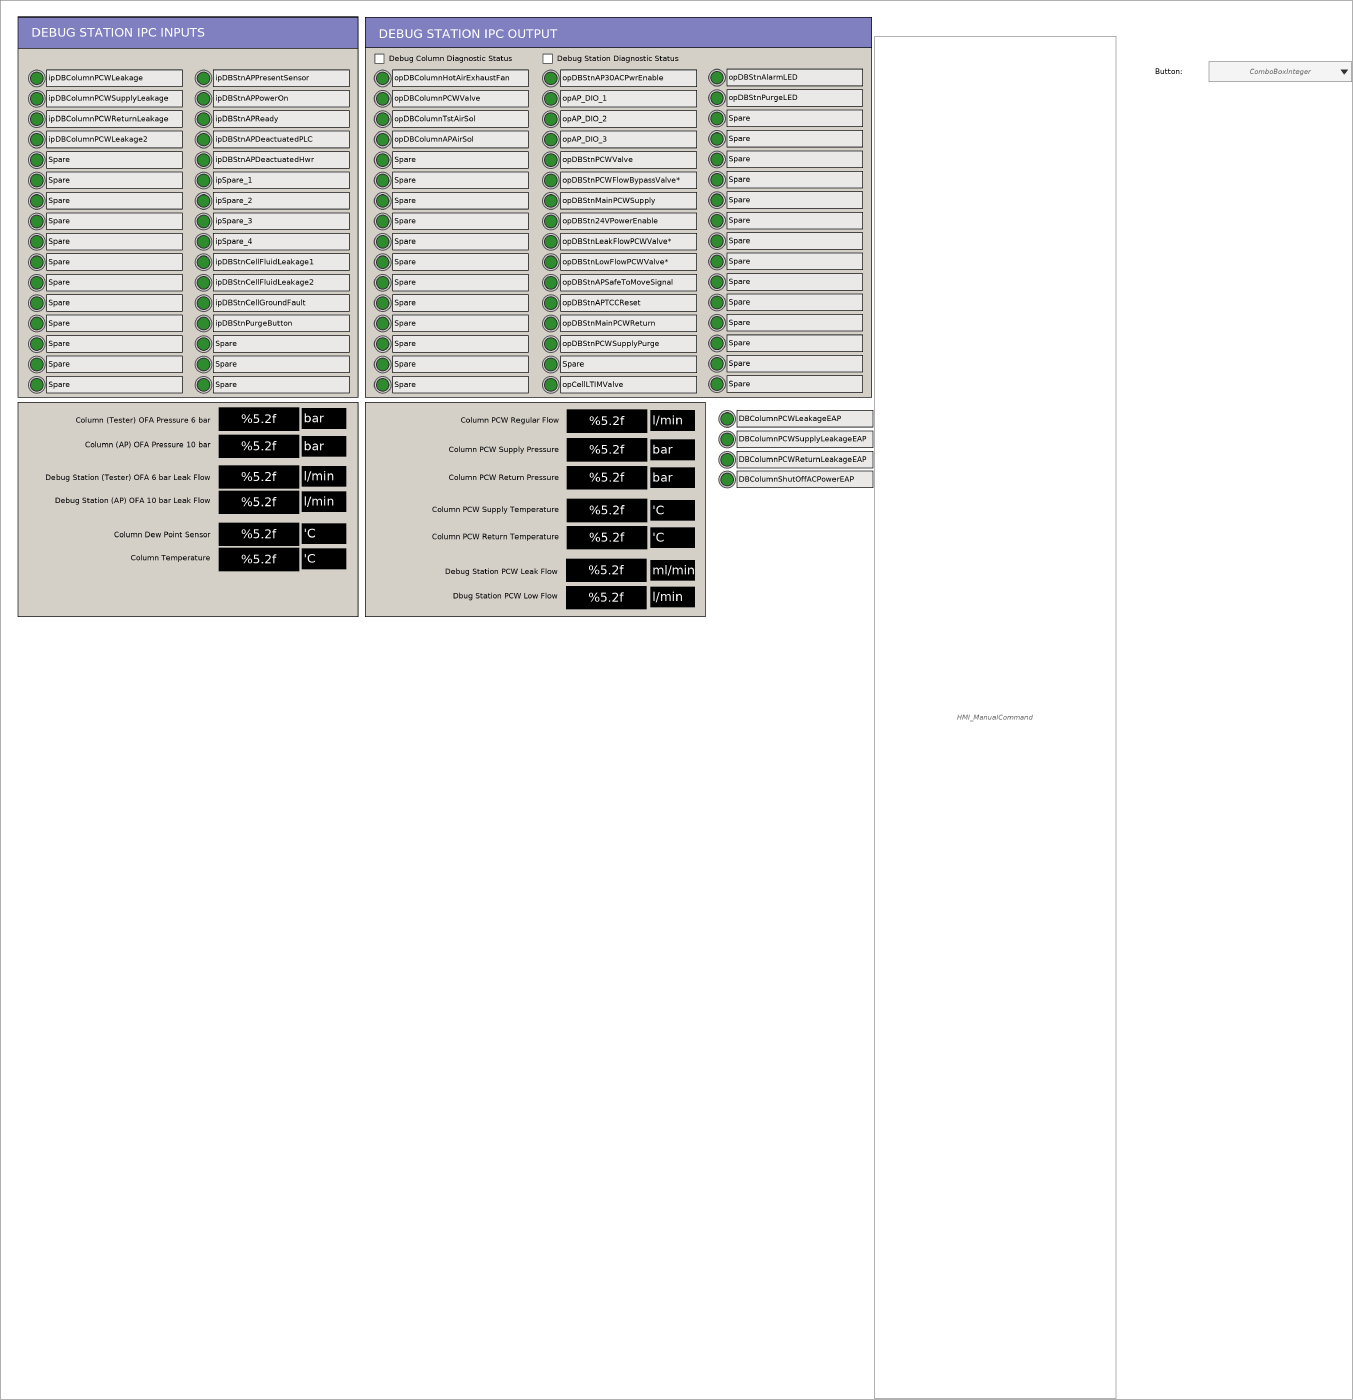
VISUALIZATION HMI_DebugStation  // 1987x2055
    Rectangle (536,590 500x315)
    Rectangle (26,590 500x315)
    Rectangle (536,42 744x541)
    Rectangle (536,25 744x45)
    Label (553,30 500x40), "DEBUG STATION IPC OUTPUT"
    Rectangle (26,24 500x559)
    Rectangle (26,25 500x46)
    Label (43,28 500x40), "DEBUG STATION IPC INPUTS"
    RoundedRectangle (68,102 200x25), "ipDBColumnPCWLeakage"
    Lamp1 (39,100 30x30), variable: fbDebugColumn.stDebugColumnDIO.ipDBColumnPCWLeakage, style: Lamp-Lamp1-Green
    RoundedRectangle (576,102 200x25), "opDBColumnHotAirExhaustFan"
        toggle fbDebugColumn.stDebugColumnDIO.opDBColumnHotAirExhaustFan
    Lamp1 (547,100 30x30), variable: fbDebugColumn.stDebugColumnDIO.opDBColumnHotAirExhaustFan, style: Lamp-Lamp1-Green
    RoundedRectangle (68,132 200x25), "ipDBColumnPCWSupplyLeakage"
    Lamp1 (39,130 30x30), variable: fbDebugColumn.stDebugColumnDIO.ipDBColumnPCWSupplyLeakage, style: Lamp-Lamp1-Green
    RoundedRectangle (68,162 200x25), "ipDBColumnPCWReturnLeakage"
    Lamp1 (39,160 30x30), variable: fbDebugColumn.stDebugColumnDIO.ipDBColumnPCWReturnLeakage, style: Lamp-Lamp1-Green
    RoundedRectangle (68,192 200x25), "ipDBColumnPCWLeakage2"
    Lamp1 (39,190 30x30), variable: fbDebugColumn.stDebugColumnDIO.ipDBColumnPCWLeakage2, style: Lamp-Lamp1-Green
    RoundedRectangle (68,222 200x25), "Spare"
    Lamp1 (39,220 30x30), style: Lamp-Lamp1-Green
    RoundedRectangle (68,252 200x25), "Spare"
    Lamp1 (39,250 30x30), style: Lamp-Lamp1-Green
    RoundedRectangle (68,282 200x25), "Spare"
    Lamp1 (39,280 30x30), style: Lamp-Lamp1-Green
    RoundedRectangle (68,312 200x25), "Spare"
    Lamp1 (39,310 30x30), style: Lamp-Lamp1-Green
    RoundedRectangle (68,342 200x25), "Spare"
    Lamp1 (39,340 30x30), style: Lamp-Lamp1-Green
    RoundedRectangle (68,372 200x25), "Spare"
    Lamp1 (39,370 30x30), style: Lamp-Lamp1-Green
    RoundedRectangle (68,402 200x25), "Spare"
    Lamp1 (39,400 30x30), style: Lamp-Lamp1-Green
    RoundedRectangle (68,432 200x25), "Spare"
    Lamp1 (39,430 30x30), style: Lamp-Lamp1-Green
    RoundedRectangle (68,462 200x25), "Spare"
    Lamp1 (39,460 30x30), style: Lamp-Lamp1-Green
    RoundedRectangle (68,492 200x25), "Spare"
    Lamp1 (39,490 30x30), style: Lamp-Lamp1-Green
    RoundedRectangle (68,522 200x25), "Spare"
    Lamp1 (39,520 30x30), style: Lamp-Lamp1-Green
    RoundedRectangle (68,552 200x25), "Spare"
    Lamp1 (39,550 30x30), style: Lamp-Lamp1-Green
    RoundedRectangle (576,132 200x25), "opDBColumnPCWValve"
        toggle fbDebugColumn.stDebugColumnDIO.opDBColumnPCWValve
    Lamp1 (547,130 30x30), variable: fbDebugColumn.stDebugColumnDIO.opDBColumnPCWValve, style: Lamp-Lamp1-Green
    RoundedRectangle (576,162 200x25), "opDBColumnTstAirSol"
        toggle fbDebugColumn.stDebugColumnDIO.opDBColumnTstAirSol
    Lamp1 (547,160 30x30), variable: fbDebugColumn.stDebugColumnDIO.opDBColumnTstAirSol, style: Lamp-Lamp1-Green
    RoundedRectangle (576,192 200x25), "opDBColumnAPAirSol"
        toggle fbDebugColumn.stDebugColumnDIO.opDBColumnAPAirSol
    Lamp1 (547,190 30x30), variable: fbDebugColumn.stDebugColumnDIO.opDBColumnAPAirSol, style: Lamp-Lamp1-Green
    RoundedRectangle (576,222 200x25), "Spare"
    Lamp1 (547,220 30x30), style: Lamp-Lamp1-Green
    RoundedRectangle (576,252 200x25), "Spare"
    Lamp1 (547,250 30x30), style: Lamp-Lamp1-Green
    RoundedRectangle (576,282 200x25), "Spare"
    Lamp1 (547,280 30x30), style: Lamp-Lamp1-Green
    RoundedRectangle (576,312 200x25), "Spare"
    Lamp1 (547,310 30x30), style: Lamp-Lamp1-Green
    RoundedRectangle (576,342 200x25), "Spare"
    Lamp1 (547,340 30x30), style: Lamp-Lamp1-Green
    RoundedRectangle (576,372 200x25), "Spare"
    Lamp1 (547,370 30x30), style: Lamp-Lamp1-Green
    RoundedRectangle (576,402 200x25), "Spare"
    Lamp1 (547,400 30x30), style: Lamp-Lamp1-Green
    RoundedRectangle (576,432 200x25), "Spare"
    Lamp1 (547,430 30x30), style: Lamp-Lamp1-Green
    RoundedRectangle (576,462 200x25), "Spare"
    Lamp1 (547,460 30x30), style: Lamp-Lamp1-Green
    RoundedRectangle (576,492 200x25), "Spare"
    Lamp1 (547,490 30x30), style: Lamp-Lamp1-Green
    RoundedRectangle (576,522 200x25), "Spare"
    Lamp1 (547,520 30x30), style: Lamp-Lamp1-Green
    RoundedRectangle (576,552 200x25), "Spare"
    Lamp1 (547,550 30x30), style: Lamp-Lamp1-Green
    RoundedRectangle (313,102 200x25), "ipDBStnAPPresentSensor"
    Lamp1 (284,100 30x30), variable: stDebugStation.fbDBStnSeq.stDebugStationDIO.ipDBStnAPPresentSensor, style: Lamp-Lamp1-Green
    RoundedRectangle (313,132 200x25), "ipDBStnAPPowerOn"
    Lamp1 (284,130 30x30), variable: stDebugStation.fbDBStnSeq.stDebugStationDIO.ipDBStnAPPowerOn, style: Lamp-Lamp1-Green
    RoundedRectangle (313,162 200x25), "ipDBStnAPReady"
    Lamp1 (284,160 30x30), variable: stDebugStation.fbDBStnSeq.stDebugStationDIO.ipDBStnAPReady, style: Lamp-Lamp1-Green
    RoundedRectangle (313,192 200x25), "ipDBStnAPDeactuatedPLC"
    Lamp1 (284,190 30x30), variable: stDebugStation.fbDBStnSeq.stDebugStationDIO.ipDBStnHandlerSafeToEnterPLC, style: Lamp-Lamp1-Green
    RoundedRectangle (313,222 200x25), "ipDBStnAPDeactuatedHwr"
    Lamp1 (284,220 30x30), variable: stDebugStation.fbDBStnSeq.stDebugStationDIO.ipDBStnHandlerSafeToEnterHwr, style: Lamp-Lamp1-Green
    RoundedRectangle (313,252 200x25), "ipSpare_1"
    Lamp1 (284,250 30x30), variable: stDebugStation.fbDBStnSeq.stDebugStationDIO.ipSpare_1, style: Lamp-Lamp1-Green
    RoundedRectangle (313,282 200x25), "ipSpare_2"
    Lamp1 (284,280 30x30), variable: stDebugStation.fbDBStnSeq.stDebugStationDIO.ipSpare_2, style: Lamp-Lamp1-Green
    RoundedRectangle (313,312 200x25), "ipSpare_3"
    Lamp1 (284,310 30x30), variable: stDebugStation.fbDBStnSeq.stDebugStationDIO.ipSpare_3, style: Lamp-Lamp1-Green
    RoundedRectangle (313,342 200x25), "ipSpare_4"
    Lamp1 (284,340 30x30), variable: stDebugStation.fbDBStnSeq.stDebugStationDIO.ipSpare_4, style: Lamp-Lamp1-Green
    RoundedRectangle (313,372 200x25), "ipDBStnCellFluidLeakage1"
    Lamp1 (284,370 30x30), variable: stDebugStation.fbDBStnSeq.stDebugStationDIO.ipDBStnCellFluidLeakage1, style: Lamp-Lamp1-Green
    RoundedRectangle (313,402 200x25), "ipDBStnCellFluidLeakage2"
    Lamp1 (284,400 30x30), variable: stDebugStation.fbDBStnSeq.stDebugStationDIO.ipDBStnCellFluidLeakage2, style: Lamp-Lamp1-Green
    RoundedRectangle (313,432 200x25), "ipDBStnCellGroundFault"
    Lamp1 (284,430 30x30), variable: stDebugStation.fbDBStnSeq.stDebugStationDIO.ipDBStnCellGroundFault, style: Lamp-Lamp1-Green
    RoundedRectangle (313,462 200x25), "ipDBStnPurgeButton"
    Lamp1 (284,460 30x30), variable: stDebugStation.fbDBStnSeq.stDebugStationDIO.ipDBStnPurgeButton, style: Lamp-Lamp1-Green
    RoundedRectangle (313,492 200x25), "Spare"
    Lamp1 (284,490 30x30), style: Lamp-Lamp1-Green
    RoundedRectangle (313,522 200x25), "Spare"
    Lamp1 (284,520 30x30), style: Lamp-Lamp1-Green
    RoundedRectangle (313,552 200x25), "Spare"
    Lamp1 (284,550 30x30), style: Lamp-Lamp1-Green
    RoundedRectangle (823,102 200x25), "opDBStnAP30ACPwrEnable"
        toggle stDebugStation.fbDBStnSeq.stDebugStationDIO.opDBStnAP240ACPwrEnable
    Lamp1 (794,100 30x30), variable: stDebugStation.fbDBStnSeq.stDebugStationDIO.opDBStnAP240ACPwrEnable, style: Lamp-Lamp1-Green
    RoundedRectangle (823,132 200x25), "opAP_DIO_1"
        toggle stDebugStation.fbDBStnSeq.stDebugStationDIO.opAP_DIO_1
    Lamp1 (794,130 30x30), variable: stDebugStation.fbDBStnSeq.stDebugStationDIO.opAP_DIO_1, style: Lamp-Lamp1-Green
    RoundedRectangle (823,162 200x25), "opAP_DIO_2"
        toggle stDebugStation.fbDBStnSeq.stDebugStationDIO.opAP_DIO_2
    Lamp1 (794,160 30x30), variable: stDebugStation.fbDBStnSeq.stDebugStationDIO.opAP_DIO_2, style: Lamp-Lamp1-Green
    RoundedRectangle (823,192 200x25), "opAP_DIO_3"
        toggle stDebugStation.fbDBStnSeq.stDebugStationDIO.opAP_DIO_3
    Lamp1 (794,190 30x30), variable: stDebugStation.fbDBStnSeq.stDebugStationDIO.opAP_DIO_3, style: Lamp-Lamp1-Green
    RoundedRectangle (823,222 200x25), "opDBStnPCWValve"
        toggle stDebugStation.fbDBStnSeq.stDebugStationDIO.opDBStnPCWValve
    Lamp1 (794,220 30x30), variable: stDebugStation.fbDBStnSeq.stDebugStationDIO.opDBStnPCWValve, style: Lamp-Lamp1-Green
    RoundedRectangle (823,252 200x25), "opDBStnPCWFlowBypassValve*"
        toggle stDebugStation.fbDBStnSeq.stDebugStationDIO.opDBStnPCWFlowBypassValve
    Lamp1 (794,250 30x30), variable: stDebugStation.fbDBStnSeq.stDebugStationDIO.opDBStnPCWFlowBypassValve, style: Lamp-Lamp1-Green
    RoundedRectangle (823,282 200x25), "opDBStnMainPCWSupply"
        toggle stDebugStation.fbDBStnSeq.stDebugStationDIO.opDBStnBypassAPAirSupplySol
    Lamp1 (794,280 30x30), variable: stDebugStation.fbDBStnSeq.stDebugStationDIO.opDBStnBypassAPAirSupplySol, style: Lamp-Lamp1-Green
    RoundedRectangle (823,312 200x25), "opDBStn24VPowerEnable"
        toggle stDebugStation.fbDBStnSeq.stDebugStationDIO.opDBStn24VPowerEnable
    Lamp1 (794,310 30x30), variable: stDebugStation.fbDBStnSeq.stDebugStationDIO.opDBStn24VPowerEnable, style: Lamp-Lamp1-Green
    RoundedRectangle (823,342 200x25), "opDBStnLeakFlowPCWValve*"
        toggle stDebugStation.fbDBStnSeq.stDebugStationDIO.opDBStnLeakFlowPCWValve
    Lamp1 (794,340 30x30), variable: stDebugStation.fbDBStnSeq.stDebugStationDIO.opDBStnLeakFlowPCWValve, style: Lamp-Lamp1-Green
    RoundedRectangle (823,372 200x25), "opDBStnLowFlowPCWValve*"
        toggle stDebugStation.fbDBStnSeq.stDebugStationDIO.opDBStnLowFlowPCWValve
    Lamp1 (794,370 30x30), variable: stDebugStation.fbDBStnSeq.stDebugStationDIO.opDBStnLowFlowPCWValve, style: Lamp-Lamp1-Green
    RoundedRectangle (823,402 200x25), "opDBStnAPSafeToMoveSignal"
        toggle stDebugStation.fbDBStnSeq.stDebugStationDIO.opDBStnAPSafeToEngage
    Lamp1 (794,400 30x30), variable: stDebugStation.fbDBStnSeq.stDebugStationDIO.opDBStnAPSafeToEngage, style: Lamp-Lamp1-Green
    RoundedRectangle (823,432 200x25), "opDBStnAPTCCReset"
        toggle stDebugStation.fbDBStnSeq.stDebugStationDIO.opDBStnAPTCCReset
    Lamp1 (794,430 30x30), variable: stDebugStation.fbDBStnSeq.stDebugStationDIO.opDBStnAPTCCReset, style: Lamp-Lamp1-Green
    RoundedRectangle (823,462 200x25), "opDBStnMainPCWReturn"
        toggle stDebugStation.fbDBStnSeq.stDebugStationDIO.opDBStnMainPCWReturn
    Lamp1 (794,460 30x30), variable: stDebugStation.fbDBStnSeq.stDebugStationDIO.opDBStnMainPCWReturn, style: Lamp-Lamp1-Green
    RoundedRectangle (823,492 200x25), "opDBStnPCWSupplyPurge"
        toggle stDebugStation.fbDBStnSeq.stDebugStationDIO.opDBStnPCWSupplyPurge
    Lamp1 (794,490 30x30), variable: stDebugStation.fbDBStnSeq.stDebugStationDIO.opDBStnPCWSupplyPurge, style: Lamp-Lamp1-Green
    RoundedRectangle (823,522 200x25), "Spare"
    Lamp1 (794,520 30x30), style: Lamp-Lamp1-Green
    RoundedRectangle (823,552 200x25), "opCellLTIMValve"
        toggle stDebugStation.fbDBStnSeq.stDebugStationDIO.opCellLTIMValve
    Lamp1 (794,550 30x30), variable: stDebugStation.fbDBStnSeq.stDebugStationDIO.opCellLTIMValve, style: Lamp-Lamp1-Green
    Textfield (320,597 120x36), "%5.2f", text variable: fbDebugColumn.stDebugColumnDIO.ipDBColumnTstAirPressure, input disabled if: TRUE
    Textfield (320,637 120x36), "%5.2f", text variable: fbDebugColumn.stDebugColumnDIO.ipDBColumnAPAirPressure, input disabled if: TRUE
    Textfield (320,682 120x36), "%5.2f", text variable: stDebugStation.fbDBStnSeq.stDebugStationDIO.ipDBStnTstAirLeakFlowSensor, input disabled if: TRUE
    Textfield (320,719 120x36), "%5.2f", text variable: stDebugStation.fbDBStnSeq.stDebugStationDIO.ipDBStnAPAirLeakFlowSensor, input disabled if: TRUE
    Label (51,686 261x30), "Debug Station (Tester) OFA 6 bar Leak Flow"
    Label (44,720 268x30), "Debug Station (AP) OFA 10 bar Leak Flow"
    Label (60,602 252x30), "Column (Tester) OFA Pressure 6 bar"
    Label (81,638 231x30), "Column (AP) OFA Pressure 10 bar"
    Textfield (830,819 120x36), "%5.2f", text variable: stDebugStation.fbDBStnSeq.stDebugStationDIO.ipDBStnPCWLeakFlowSensor, input disabled if: TRUE
    Textfield (830,859 120x36), "%5.2f", text variable: stDebugStation.fbDBStnSeq.stDebugStationDIO.ipDBStnPCWLowFlowSensor, input disabled if: TRUE
    Label (620,824 202x30), "Debug Station PCW Leak Flow"
    Label (574,860 248x30), "Dbug Station PCW Low Flow"
    Textfield (831,771 120x36), "%5.2f", text variable: fbDebugColumn.stDebugColumnDIO.ipDBColumnPCWReturnTemperature, input disabled if: TRUE
    Textfield (831,683 120x36), "%5.2f", text variable: fbDebugColumn.stDebugColumnDIO.ipDBColumnPCWReturnPressure, input disabled if: TRUE
    Textfield (831,600 120x36), "%5.2f", text variable: fbDebugColumn.stDebugColumnDIO.ipDBColumnPCWRegularFlowSensor, input disabled if: TRUE
    Textfield (831,642 120x36), "%5.2f", text variable: fbDebugColumn.stDebugColumnDIO.ipDBColumnPCWSupplyPressure, input disabled if: TRUE
    Textfield (831,731 120x36), "%5.2f", text variable: fbDebugColumn.stDebugColumnDIO.ipDBColumnPCWSupplyTemperature, input disabled if: TRUE
    Label (613,602 211x30), "Column PCW Regular Flow"
    Label (616,645 208x30), "Column PCW Supply Pressure"
    Label (641,686 183x30), "Column PCW Return Pressure"
    Label (595,733 229x30), "Column PCW Supply Temperature"
    Label (611,773 213x30), "Column PCW Return Temperature"
    Rectangle (955,602 65x30), "l/min"
    Rectangle (955,645 65x30), "bar"
    Rectangle (955,686 65x30), "bar"
    Rectangle (955,734 65x30), "'C"
    Rectangle (955,774 65x30), "'C"
    Rectangle (955,822 65x30), "ml/min"
    Rectangle (955,861 65x30), "l/min"
    Rectangle (443,599 65x30), "bar"
    Rectangle (443,640 65x30), "bar"
    Rectangle (443,684 65x30), "l/min"
    Rectangle (443,721 65x30), "l/min"
    Textfield (320,766 120x36), "%5.2f", text variable: fbDebugColumn.stDebugColumnDIO.ipDBColumnDewPointSensor, input disabled if: TRUE
    Textfield (320,803 120x36), "%5.2f", text variable: fbDebugColumn.stDebugColumnDIO.ipDBColumnTempSensor, input disabled if: TRUE
    Label (133,770 179x30), "Column Dew Point Sensor"
    Label (162,804 150x30), "Column Temperature"
    Rectangle (443,768 65x30), "'C"
    Rectangle (443,805 65x30), "'C"
    Checkbox (795,71 224x30), "Debug Station Diagnostic Status", variable: stDebugStation.fbDBStnSeq.stDebugStationVIO.bDiagnosticMode
    Checkbox (548,71 222x30), "Debug Column Diagnostic Status", variable: fbDebugColumn.stDebugColumnVIO.bDiagnosticMode
    RoundedRectangle (1082,602 200x25), "DBColumnPCWLeakageEAP"
        toggle fbDebugColumn.stDebugColumnDIO.eapDBColumnPCWLeakage
    Lamp1 (1053,600 30x30), variable: fbDebugColumn.stDebugColumnDIO.eapDBColumnPCWLeakage, style: Lamp-Lamp1-Green
    RoundedRectangle (1082,632 200x25), "DBColumnPCWSupplyLeakageEAP"
        toggle fbDebugColumn.stDebugColumnDIO.eapDBColumnPCWSupplyLeakage
    Lamp1 (1053,630 30x30), variable: fbDebugColumn.stDebugColumnDIO.eapDBColumnPCWSupplyLeakage, style: Lamp-Lamp1-Green
    RoundedRectangle (1082,662 200x25), "DBColumnPCWReturnLeakageEAP"
        toggle fbDebugColumn.stDebugColumnDIO.eapDBColumnPCWReturnLeakage
    Lamp1 (1053,660 30x30), variable: fbDebugColumn.stDebugColumnDIO.eapDBColumnPCWReturnLeakage, style: Lamp-Lamp1-Green
    Frame (1284,53 355x2000), invisible if: Not bEnableManualCommandTest1 AND Not bEnableManualCommandTest2
        shows HMI_ManualCommand()
    Lamp1 (1038,99 30x30), variable: stDebugStation.fbDBStnSeq.stDebugStationDIO.opDBStnAlarmLED, style: Lamp-Lamp1-Green
    RoundedRectangle (1067,101 200x25), "opDBStnAlarmLED"
        toggle stDebugStation.fbDBStnSeq.stDebugStationDIO.opDBStnAlarmLED
    RoundedRectangle (1067,131 200x25), "opDBStnPurgeLED"
        toggle stDebugStation.fbDBStnSeq.stDebugStationDIO.opDBStnPurgeLED
    Lamp1 (1038,129 30x30), variable: stDebugStation.fbDBStnSeq.stDebugStationDIO.opDBStnPurgeLED, style: Lamp-Lamp1-Green
    RoundedRectangle (1067,161 200x25), "Spare"
    Lamp1 (1038,159 30x30), style: Lamp-Lamp1-Green
    RoundedRectangle (1067,191 200x25), "Spare"
    Lamp1 (1038,189 30x30), style: Lamp-Lamp1-Green
    RoundedRectangle (1067,221 200x25), "Spare"
    Lamp1 (1038,219 30x30), style: Lamp-Lamp1-Green
    RoundedRectangle (1067,251 200x25), "Spare"
    Lamp1 (1038,249 30x30), style: Lamp-Lamp1-Green
    RoundedRectangle (1067,281 200x25), "Spare"
    Lamp1 (1038,279 30x30), style: Lamp-Lamp1-Green
    RoundedRectangle (1067,311 200x25), "Spare"
    Lamp1 (1038,309 30x30), style: Lamp-Lamp1-Green
    RoundedRectangle (1067,341 200x25), "Spare"
    Lamp1 (1038,339 30x30), style: Lamp-Lamp1-Green
    RoundedRectangle (1067,371 200x25), "Spare"
    Lamp1 (1038,369 30x30), style: Lamp-Lamp1-Green
    RoundedRectangle (1067,401 200x25), "Spare"
    Lamp1 (1038,399 30x30), style: Lamp-Lamp1-Green
    RoundedRectangle (1067,431 200x25), "Spare"
    Lamp1 (1038,429 30x30), style: Lamp-Lamp1-Green
    RoundedRectangle (1067,461 200x25), "Spare"
    Lamp1 (1038,459 30x30), style: Lamp-Lamp1-Green
    RoundedRectangle (1067,491 200x25), "Spare"
    Lamp1 (1038,489 30x30), style: Lamp-Lamp1-Green
    RoundedRectangle (1067,521 200x25), "Spare"
    Lamp1 (1038,519 30x30), style: Lamp-Lamp1-Green
    RoundedRectangle (1067,551 200x25), "Spare"
    Lamp1 (1038,549 30x30), style: Lamp-Lamp1-Green
    RoundedRectangle (1082,691 200x25), "DBColumnShutOffACPowerEAP"
        toggle fbDebugColumn.stDebugColumnDIO.eapShutOffAllACPower
    Lamp1 (1053,689 30x30), variable: fbDebugColumn.stDebugColumnDIO.eapShutOffAllACPower, style: Lamp-Lamp1-Green
    ComboBoxInteger (1775,90 210x30), variable: TestManually.iBtnNo
    Label (1680,90 76x30), "Button:"
END_VISUALIZATION

(* stored: Version 1.1.0.1, ProductVersion 3.1.4022.18
   Visu HMI_DebugStation: Id {917bb58c-27c4-422a-8496-349c295d05aa} *)
